VAR_GLOBAL
	instConveyorFeedOutStackerCrane	:	FactoryIO.FB_Foerderband;
	instConveyorFeedOutTwoMeter	:	FactoryIO.FB_Foerderband;
	instConveyorFeedOutCurve	:	FactoryIO.FB_Foerderband;
	instConveyorFeedOutLong	:	FactoryIO.FB_Foerderband;
	instPartMovingOut	:	FB_RunControl;
END_VAR

(* stored: Version 1.1.0.1
   GVL ConveyorbeltsOutfeed: Id {308910a0-8f79-4f67-9fa4-29ffd7c77145} *)
